// TIA Portal V17 export
// export: Created 2025-05-22T05:59:47.0520576Z, ExportSetting WithDefaults, DisplayName Totally Integrated Automation Portal, DisplayVersion V17 Update 8, DisplayName TIA Portal Openness, DisplayVersion V17 Update 8, DisplayName TIA Portal Version Control Interface, DisplayVersion V17, DisplayName SINAMICS Startdrive Advanced, DisplayVersion V17 SP2, DisplayName SINAMICS Startdrive G110M, G120, G120C, G120D, G120P, G115D, DisplayVersion V17 SP2, DisplayName SINAMICS Startdrive G130, G150, S120, S150, SINAMICS MV, S210, DisplayVersion V17 SP2, DisplayName STEP 7 Professional, DisplayVersion V17 Update 8, DisplayName SINUMERIK ONE STEP 7 Toolbox, DisplayVersion V17 Update 12, DisplayName SINUMERIK ONE PLC Basic Program Plus, DisplayVersion V17 Update 12, DisplayName SINUMERIK 840D sl STEP 7 Toolbox, DisplayVersion V17 Update 12, DisplayName STEP 7 Safety, DisplayVersion V17 Update 6, DisplayName WinCC Advanced, DisplayVersion V17 Update 8
FUNCTION "FC8000_PART_STATUS" : Void   // FC8000, LAD
{ S7_Optimized_Access := 'FALSE' }
AUTHOR : ETXETAR
VERSION : 1.0
// BIT "PUN_A_PUN_B"
// 0 = THERE IS ONLY 1 "PUN DATA" OR "PART ID" 
// 1 = THERE ARE SEPARATE "PUN DATA" OR "PART ID" FOR PART A AND PART B
// 
// BIT "LIFTING_ONLY_1_POS"
// 0 = LIFTING HAS 2 OR 3 POSITIONS FOR AXIS W
// 1 = LIFTING HAS ONLY 1 POSITION FOR AXIS W
// stored: AutoNumber false, IsIECCheckEnabled false, SetENOAutomatically false, UDAEnableTagReadback false
   VAR_TEMP
      Workpiece_Screen : Int;
      Workpiece_Screen_selectd : Bool;
      zero : Byte;
      one : Byte;
      OPTION_ON : Bool;
      OPTION_OFF : Bool;
   END_VAR
BEGIN

REGION Network 1: OPTION OFF / OPTIONS OFF
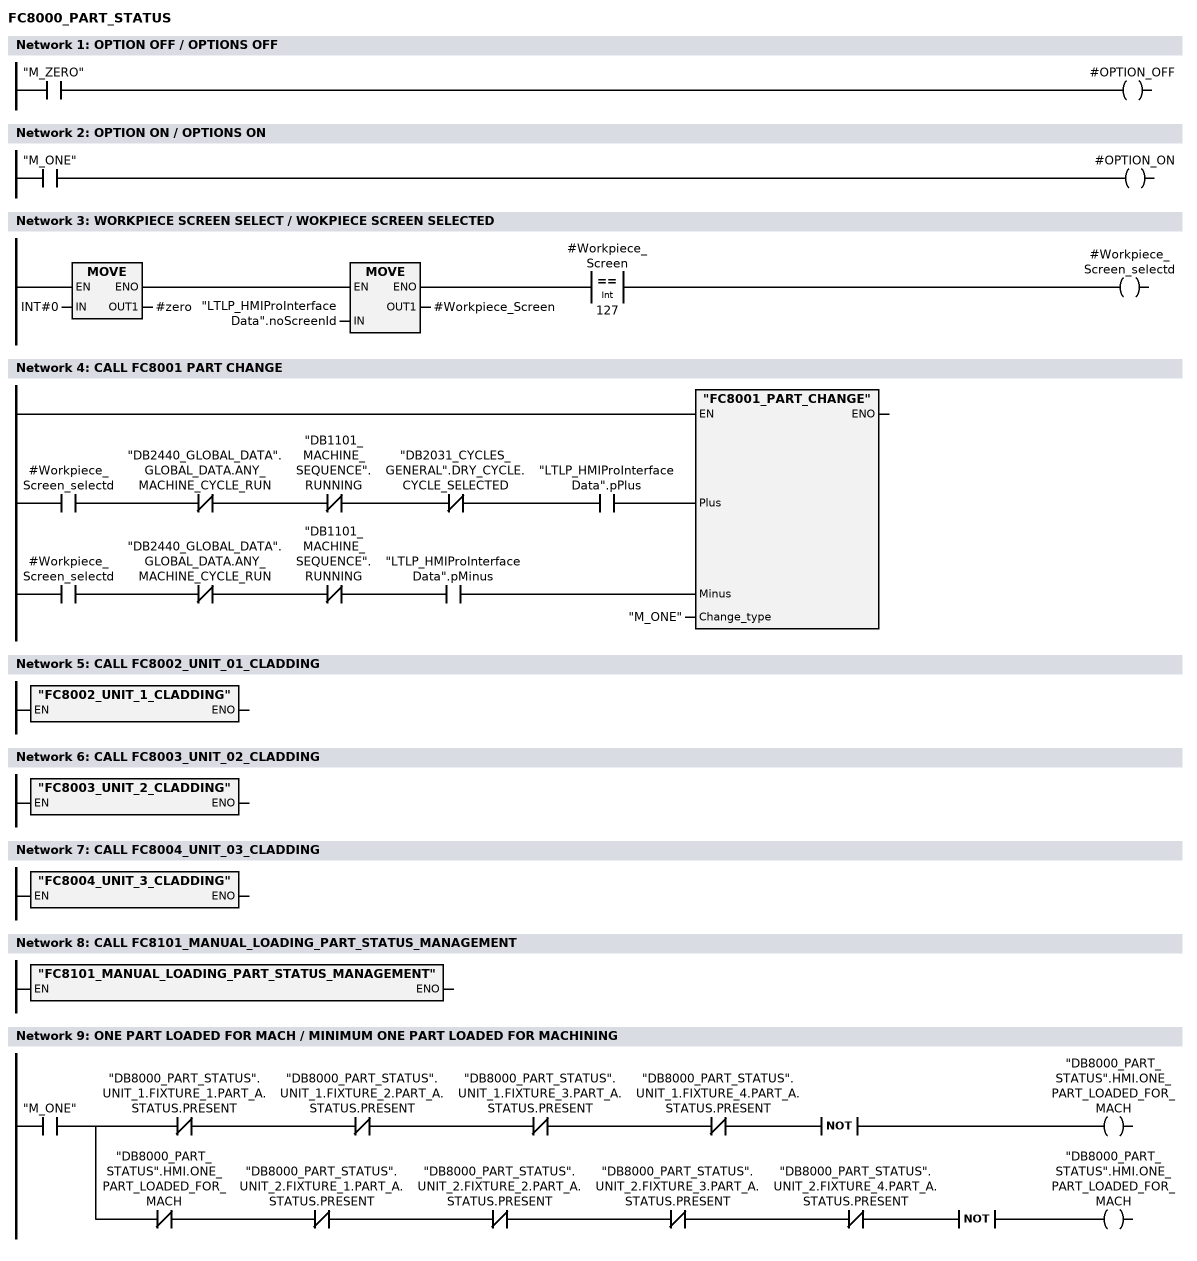
   RUNG wire#powerrail
      Contact( "M_ZERO" )
      Coil( #OPTION_OFF )
   END_RUNG
   // the same network as SCL:
   #OPTION_OFF := "M_ZERO";
END_REGION

REGION Network 2: OPTION ON / OPTIONS ON
   RUNG wire#powerrail
      Contact( "M_ONE" )
      Coil( #OPTION_ON )
   END_RUNG
   // the same network as SCL:
   #OPTION_ON := "M_ONE";
END_REGION

REGION Network 3: WORKPIECE SCREEN SELECT / WOKPIECE SCREEN SELECTED
   RUNG wire#powerrail
      { S7_GenerateENO := "TRUE" } Move(in := INT#0, out1 => #zero)
      { S7_GenerateENO := "TRUE" } Move(in := "LTLP_HMIProInterfaceData".noScreenId, out1 => #Workpiece_Screen)
      { S7_Templates := "SrcType := Int" } EQ_Contact(in1 := #Workpiece_Screen, in2 := 127)
      Coil( #Workpiece_Screen_selectd )
   END_RUNG
   // the same network as SCL:
   // ENO of a box is taken as its EN; it also drops when the box reports an error
   #zero := INT#0;
   #Workpiece_Screen := "LTLP_HMIProInterfaceData".noScreenId;
   #Workpiece_Screen_selectd := #Workpiece_Screen = 127;
END_REGION

REGION Network 4: CALL FC8001 PART CHANGE
   RUNG wire#powerrail
      "FC8001_PART_CHANGE"(Plus := wire#w1, Minus := wire#w2, Change_type := "M_ONE")
   END_RUNG
   RUNG wire#powerrail
      Contact( #Workpiece_Screen_selectd )
      I_Contact( "DB2440_GLOBAL_DATA".GLOBAL_DATA.ANY_MACHINE_CYCLE_RUN )
      I_Contact( "DB1101_MACHINE_SEQUENCE".RUNNING )
      I_Contact( "DB2031_CYCLES_GENERAL".DRY_CYCLE.CYCLE_SELECTED )
      Contact( "LTLP_HMIProInterfaceData".pPlus )
   END_RUNG wire#w1
   RUNG wire#powerrail
      Contact( #Workpiece_Screen_selectd )
      I_Contact( "DB2440_GLOBAL_DATA".GLOBAL_DATA.ANY_MACHINE_CYCLE_RUN )
      I_Contact( "DB1101_MACHINE_SEQUENCE".RUNNING )
      Contact( "LTLP_HMIProInterfaceData".pMinus )
   END_RUNG wire#w2
   // the same network as SCL:
   "FC8001_PART_CHANGE"(Plus := #Workpiece_Screen_selectd AND NOT "DB2440_GLOBAL_DATA".GLOBAL_DATA.ANY_MACHINE_CYCLE_RUN AND NOT "DB1101_MACHINE_SEQUENCE".RUNNING AND NOT "DB2031_CYCLES_GENERAL".DRY_CYCLE.CYCLE_SELECTED AND "LTLP_HMIProInterfaceData".pPlus,
                        Minus := #Workpiece_Screen_selectd AND NOT "DB2440_GLOBAL_DATA".GLOBAL_DATA.ANY_MACHINE_CYCLE_RUN AND NOT "DB1101_MACHINE_SEQUENCE".RUNNING AND "LTLP_HMIProInterfaceData".pMinus,
                        Change_type := "M_ONE");
END_REGION

REGION Network 5: CALL FC8002_UNIT_01_CLADDING
   RUNG wire#powerrail
      "FC8002_UNIT_1_CLADDING"()
   END_RUNG
   // the same network as SCL:
   "FC8002_UNIT_1_CLADDING"();
END_REGION

REGION Network 6: CALL FC8003_UNIT_02_CLADDING
   RUNG wire#powerrail
      "FC8003_UNIT_2_CLADDING"()
   END_RUNG
   // the same network as SCL:
   "FC8003_UNIT_2_CLADDING"();
END_REGION

REGION Network 7: CALL FC8004_UNIT_03_CLADDING
   RUNG wire#powerrail
      "FC8004_UNIT_3_CLADDING"()
   END_RUNG
   // the same network as SCL:
   "FC8004_UNIT_3_CLADDING"();
END_REGION

REGION Network 8: CALL FC8101_MANUAL_LOADING_PART_STATUS_MANAGEMENT
   RUNG wire#powerrail
      "FC8101_MANUAL_LOADING_PART_STATUS_MANAGEMENT"()
   END_RUNG
   // the same network as SCL:
   "FC8101_MANUAL_LOADING_PART_STATUS_MANAGEMENT"();
END_REGION

REGION Network 9: ONE PART LOADED FOR MACH / MINIMUM ONE PART LOADED FOR MACHINING
   RUNG wire#powerrail
      Contact( "M_ONE" )
      wire#w1
      I_Contact( "DB8000_PART_STATUS".UNIT_1.FIXTURE_1.PART_A.STATUS.PRESENT )
      I_Contact( "DB8000_PART_STATUS".UNIT_1.FIXTURE_2.PART_A.STATUS.PRESENT )
      I_Contact( "DB8000_PART_STATUS".UNIT_1.FIXTURE_3.PART_A.STATUS.PRESENT )
      I_Contact( "DB8000_PART_STATUS".UNIT_1.FIXTURE_4.PART_A.STATUS.PRESENT )
      Not()
      Coil( "DB8000_PART_STATUS".HMI.ONE_PART_LOADED_FOR_MACH )
   END_RUNG
   RUNG wire#w1
      I_Contact( "DB8000_PART_STATUS".HMI.ONE_PART_LOADED_FOR_MACH )
      I_Contact( "DB8000_PART_STATUS".UNIT_2.FIXTURE_1.PART_A.STATUS.PRESENT )
      I_Contact( "DB8000_PART_STATUS".UNIT_2.FIXTURE_2.PART_A.STATUS.PRESENT )
      I_Contact( "DB8000_PART_STATUS".UNIT_2.FIXTURE_3.PART_A.STATUS.PRESENT )
      I_Contact( "DB8000_PART_STATUS".UNIT_2.FIXTURE_4.PART_A.STATUS.PRESENT )
      Not()
      Coil( "DB8000_PART_STATUS".HMI.ONE_PART_LOADED_FOR_MACH )
   END_RUNG
   // the same network as SCL:
   "DB8000_PART_STATUS".HMI.ONE_PART_LOADED_FOR_MACH := NOT ("M_ONE" AND NOT "DB8000_PART_STATUS".UNIT_1.FIXTURE_1.PART_A.STATUS.PRESENT AND NOT "DB8000_PART_STATUS".UNIT_1.FIXTURE_2.PART_A.STATUS.PRESENT AND NOT "DB8000_PART_STATUS".UNIT_1.FIXTURE_3.PART_A.STATUS.PRESENT AND NOT "DB8000_PART_STATUS".UNIT_1.FIXTURE_4.PART_A.STATUS.PRESENT);
   "DB8000_PART_STATUS".HMI.ONE_PART_LOADED_FOR_MACH := NOT ("M_ONE" AND NOT "DB8000_PART_STATUS".HMI.ONE_PART_LOADED_FOR_MACH AND NOT "DB8000_PART_STATUS".UNIT_2.FIXTURE_1.PART_A.STATUS.PRESENT AND NOT "DB8000_PART_STATUS".UNIT_2.FIXTURE_2.PART_A.STATUS.PRESENT AND NOT "DB8000_PART_STATUS".UNIT_2.FIXTURE_3.PART_A.STATUS.PRESENT AND NOT "DB8000_PART_STATUS".UNIT_2.FIXTURE_4.PART_A.STATUS.PRESENT);
END_REGION
END_FUNCTION
